FUNCTION_BLOCK T_UnitTestUnderTest EXTENDS T_UnitTestBase
VAR_INPUT
END_VAR
VAR_OUTPUT
END_VAR
VAR
END_VAR

END_FUNCTION_BLOCK

(* stored: Version 1.1.0.1, ProductVersion 3.1.4024.4
   POU T_UnitTestUnderTest: Id {7bfed642-dce0-402f-827d-e5704a2c4489}, SpecialFunc None *)
